// TIA Portal V21 export
DATA_BLOCK "AlarmsLogic_DB"   // DB202
{ S7_Optimized_Access := 'TRUE'; DB_Accessible_From_OPC_UA := 'FALSE' }
// stored: AutoNumber false, DBAccessibleFromOPCUA false, DBAccessibleFromWebserver false, MemoryReserve 100
BEGIN
END_DATA_BLOCK
